// TwinCAT 3 PLC project CCSSimulator
// ProgramVersion: 3.1.4023.0
// libraries:
//   ESO CCS PLC Library, * (ccsim)
//   ESO LDC Timer Library, * (ESO)
//   Tc2_Standard, * (Beckhoff Automation GmbH)
//   Tc2_System, * (Beckhoff Automation GmbH)
//   Tc3_Module, * (Beckhoff Automation GmbH)
//   VisuDialogs, * (System)
// project tree:
//   / GlobalTextList.TcGTLO, PlcTask.TcTTO (not stored), Visualization Manager.TcVMO (not stored)
//   POUs/ MAIN.TcPOU
//   VISUs/ GUI_CCS_SIM.TcVIS (not stored), GUI_TIMER.TcVIS (not stored)
// real-time tasks:
//   TASK PlcTask: cycle T#10ms, priority 20, ADS port 350
//   TASK FastTask: cycle T#50000us, priority 1, ADS port 351
//   TASK SlowTask: cycle T#100000us, priority 2, ADS port 352
// I/O:
//   DEVICE Device 1 (RT-Ethernet Adapter)
// variable links:
//   CCSSimulator/CCSSimulator Instance <-> TcCOM Objects/Object1 (TcNtpExternalTimeProvider)
//     PlcTask Inputs/MAIN.fbTimer.i_exNtpConnected <-> Diagnostic/bIsConnected
//     PlcTask Inputs/MAIN.fbTimer.i_exNtpExtTime <-> Outputs/nExtTime
//     PlcTask Inputs/MAIN.fbTimer.i_exNtpSynchronized <-> Diagnostic/bIsSynchronized
//     PlcTask Inputs/MAIN.fbTimer.i_exNtpSysTime <-> Outputs/nSysTime
//   CCSSimulator/CCSSimulator Instance <-> TcCOM Objects/Object2 (trkParams)
//     PlcTask Outputs/MAIN.ccs_sim.q_ccs_data <-> Inputs/CcsData
//     PlcTask Outputs/MAIN.fbTimer.q_timeInfo <-> Inputs/TimeInfo
//   CCSSimulator/CCSSimulator Instance <-> TcCOM Objects/Object3 (trkModule)
//     PlcTask Inputs/MAIN.ccs_sim.i_trk_data <-> Outputs/TrackingData
//     PlcTask Outputs/MAIN.ccs_sim.q_mean_coordinates <-> Inputs/MeanCoordinates
//     PlcTask Outputs/MAIN.ccs_sim.q_mudpi_cfg <-> Inputs/MudpiConfig
//     PlcTask Outputs/MAIN.fbTimer.q_timeInfo <-> Inputs/TimeInfo
//   TcCOM Objects/Object2 (trkParams) <-> TcCOM Objects/Object3 (trkModule)
//     Outputs/SlaParams <-> Inputs/SlaParams

// ---- POUs/MAIN.TcPOU
PROGRAM MAIN
VAR
	ccs_sim:	FB_CCS_SIM;
	fbTimer: FB_TIME;
END_VAR

fbTimer();
ccs_sim();

END_PROGRAM
